FUNCTION_BLOCK TwoConCtlCentral (* Composite Function Block Type *)
  (* Standard: 61499-2 *)
  (* Version 0.2, 2003-12-05, JHC, Rockwell Automation, Renamed from NEWCOMPFB. *)
  (* Version 0.1, 2002-01-08, JHC, Rockwell Automation, Added DLY FB as example. *)
  (* Version 0.0, 2000-05-27, JHC, Rockwell Automation *)
  (* Compiler header: package fb.rt.conveyorIEC61499; *)
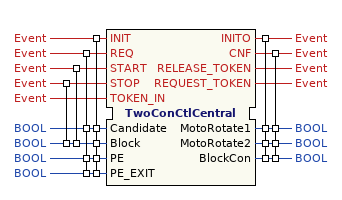
  EVENT_INPUT
    INIT WITH Candidate, Block, PE, PE_EXIT; (* Initialization Request *)
    REQ WITH Candidate, PE, PE_EXIT; (* Normal Execution Request *)
    START WITH Block;
    STOP WITH Block;
    TOKEN_IN;
  END_EVENT
  EVENT_OUTPUT
    INITO WITH MotoRotate1, MotoRotate2, BlockCon; (* Initialization Confirm *)
    CNF WITH MotoRotate1, MotoRotate2, BlockCon; (* Execution Confirmation *)
    RELEASE_TOKEN;
    REQUEST_TOKEN;
  END_EVENT
  VAR_INPUT
    Candidate : BOOL;
    Block : BOOL;
    PE : BOOL;
    PE_EXIT : BOOL;
  END_VAR
  VAR_OUTPUT
    MotoRotate1 : BOOL;
    MotoRotate2 : BOOL;
    BlockCon : BOOL;
  END_VAR
  FBS
    FC12 : ConveyorCTLCentral;
    FC11 : ConveyorCTL(PE := 0, Block := 0, Candidate := 0);
  END_FBS
  EVENT_CONNECTIONS
    START TO FC12.CAS_START;
    STOP TO FC12.CAS_STOP;
    REQ TO FC12.REQ;
    FC11.INITO TO FC12.INIT;
    FC12.INITO TO INITO;
    FC12.CNF TO CNF;
    FC12.STOP TO FC11.CAS_STOP;
    FC12.START TO FC11.CAS_START;
    INIT TO FC11.INIT;
    REQ TO FC11.REQ;
    FC12.RequestToken TO RELEASE_TOKEN;
    FC12.RequestToken TO REQUEST_TOKEN;
    FC12.ReleaseToken TO RELEASE_TOKEN;
  END_CONNECTIONS
  DATA_CONNECTIONS
    FC11.MotoRotate TO MotoRotate1;
    FC12.MotoRotate TO MotoRotate2;
    FC12.BlockCon TO BlockCon;
    Candidate TO FC12.Candidate;
    Block TO FC12.Block;
    PE TO FC12.PE;
  END_CONNECTIONS
END_FUNCTION_BLOCK
